{attribute 'GeneratedUsingTerminal: EL9181--0000'}
{attribute addProperty BoxType "EL9181--0000"}
{attribute addProperty Description "EL9181 Potential Connection, 2 x 8 contacts"}
{attribute addProperty Physics "KK"}
{attribute addProperty Id "EL9181"}
{attribute addProperty CRC "2413040443"}
{attribute addProperty Size "0"}
TYPE EL9181_8FD4133B EXTENDS EtcSlaveTerminalBase_947E5A46 :
STRUCT
END_STRUCT
END_TYPE

(* stored: Version 1.2.0.0, ProductVersion 3.1.4024.11
   DUT EL9181_8FD4133B: Id {5e849cc4-d690-4bee-8e0c-df99bea07691} *)
